INTERFACE I_TcpIpConnection EXTENDS I_Component

{attribute 'monitoring' := 'call'}
PROPERTY ConnectionState : E_SocketConnectionState
GET
END_GET
END_PROPERTY

{attribute 'monitoring' := 'call'}
PROPERTY IP : T_IPv4Addr
SET
END_SET
END_PROPERTY

{attribute 'monitoring' := 'call'}
PROPERTY Port : UDINT
SET
END_SET
END_PROPERTY

METHOD RegisterCommand
VAR_INPUT
	Command : I_TcpIpSubscription;
END_VAR
END_METHOD

METHOD SendCommand
VAR_INPUT
	Command : POINTER TO ST_TcpIpPayload;
END_VAR
END_METHOD

METHOD SendPriorityCommand
VAR_INPUT
	Command : POINTER TO ST_TcpIpPayload;
END_VAR
END_METHOD

PROPERTY Socket : T_HSOCKET
GET
END_GET
END_PROPERTY

END_INTERFACE

(* stored: Version 1.1.0.1, ProductVersion 3.1.4026.18
   Itf I_TcpIpConnection: Id {1658d39e-d185-4358-89f1-d41dc0880621}
   Property ConnectionState: Id {b6788988-6230-4132-96cf-dbe8ae56b615}
   Get Get: Id {785a2b48-ba5e-4389-934a-e3939630aef7}
   Property IP: Id {24bd76b7-a680-438b-9d10-edebf1338460}
   Set Set: Id {4f3c0c45-bbcc-42b1-aeba-c2b36d964a6f}
   Property Port: Id {a61080ca-af12-432d-bb0d-cee6e914b428}
   Set Set: Id {0d2c351d-1561-430d-83aa-5d8f1ca8a35a}
   Method RegisterCommand: Id {2cf8e55d-0a6e-4004-903d-c0badd10454d}
   Method SendCommand: Id {00c54666-8a63-458b-b36a-68a0b1532086}
   Method SendPriorityCommand: Id {31208047-4915-41c1-8101-e562202a0c89}
   Property Socket: Id {cede5a45-bdea-4442-941b-53ecf95f45de}
   Get Get: Id {b8217d4e-78e1-4b96-8374-7bb1d0bfa02f} *)
